FUNCTION_BLOCK IORevPiAIO (* Analog I/O module for Revolution Pi by KUNBUS GmbH *)
  (* Standard: 61499-2; Description: Copyright (c) 2024 Monika Wenger This program and the accompanying materials are made available under the terms of the Eclipse Public License 2.0 which is available at https://www.eclipse.org/legal/epl-2.0/ SPDX-License-Identifier: EPL-2.0 *)
  (* Version 1.0, 2024-03-27, Monika Wenger, reconstructed from code *)
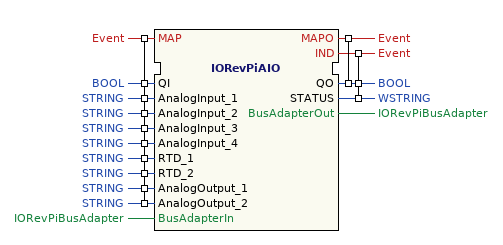
  EVENT_INPUT
    MAP WITH AnalogInput_1, AnalogInput_2, RTD_1, AnalogInput_3, AnalogInput_4, RTD_2, AnalogOutput_1, AnalogOutput_2, QI; (* Map Pins *)
  END_EVENT
  EVENT_OUTPUT
    MAPO WITH QO; (* Confirm Pin Mapping *)
    IND WITH QO, STATUS; (* Indication from Resource *)
  END_EVENT
  VAR_INPUT
    QI : BOOL; (* Event Input Qualifier *)
    AnalogInput_1 : STRING;
    AnalogInput_2 : STRING;
    AnalogInput_3 : STRING;
    AnalogInput_4 : STRING;
    RTD_1 : STRING;
    RTD_2 : STRING;
    AnalogOutput_1 : STRING;
    AnalogOutput_2 : STRING;
  END_VAR
  VAR_OUTPUT
    QO : BOOL; (* Event Output Qualifier *)
    STATUS : WSTRING; (* Service Status *)
  END_VAR
  SOCKETS
    BusAdapterIn : IORevPiBusAdapter;
  END_SOCKETS
  PLUGS
    BusAdapterOut : IORevPiBusAdapter;
  END_PLUGS
END_FUNCTION_BLOCK
